// SIMATIC S7-200 SMART project (STEP 7-Micro/WIN SMART), CPU SR40

ORGANIZATION_BLOCK MAIN:OB1
TITLE=程序注释
BEGIN
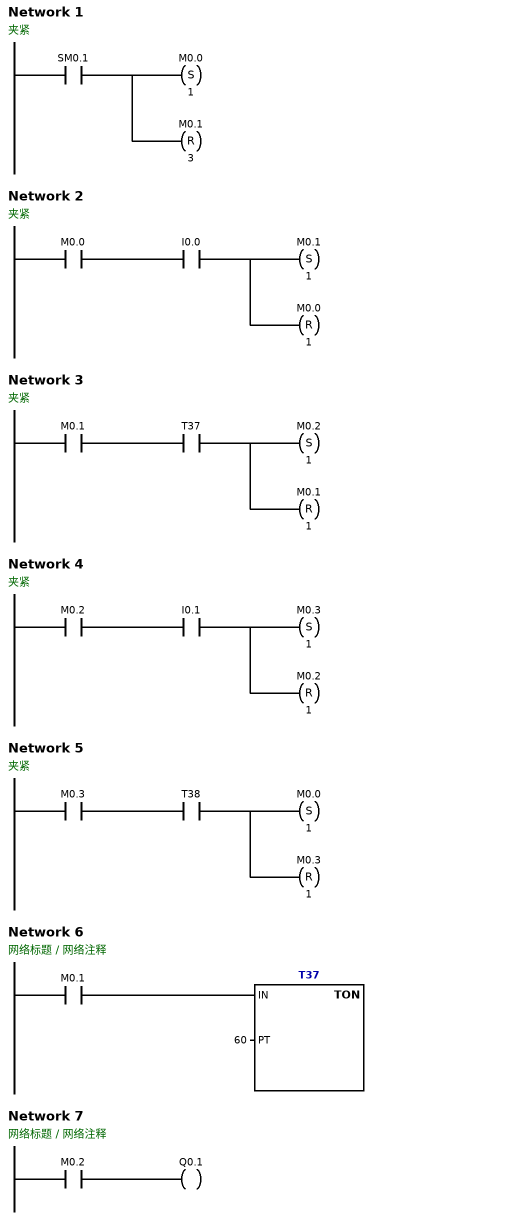
Network 1
// 夹紧
LD     SM0.1
S      M0.0, 1
R      M0.1, 3
Network 2
// 夹紧
LD     M0.0
A      I0.0
S      M0.1, 1
R      M0.0, 1
Network 3
// 夹紧
LD     M0.1
A      T37
S      M0.2, 1
R      M0.1, 1
Network 4
// 夹紧
LD     M0.2
A      I0.1
S      M0.3, 1
R      M0.2, 1
Network 5
// 夹紧
LD     M0.3
A      T38
S      M0.0, 1
R      M0.3, 1
Network 6
// 网络标题
// 网络注释
LD     M0.1
TON    T37, 60
Network 7
// 网络标题
// 网络注释
LD     M0.2
=      Q0.1
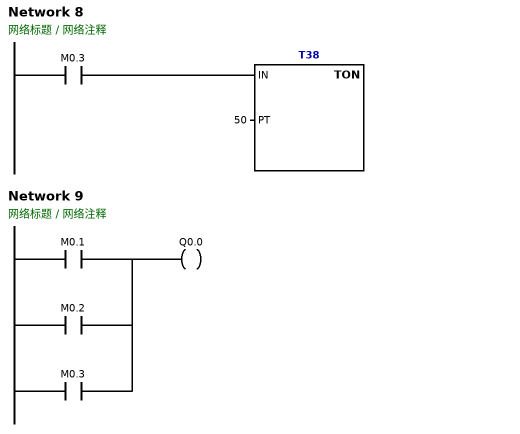
Network 8
// 网络标题
// 网络注释
LD     M0.3
TON    T38, 50
Network 9
// 网络标题
// 网络注释
LD     M0.1
O      M0.2
O      M0.3
=      Q0.0
END_ORGANIZATION_BLOCK
